// TIA Portal V20 export
DATA_BLOCK "InstShiftmodel"   // DB101
TITLE = Instanz Shiftmodel / InstanceShiftmodel
{ DB_Accessible_From_OPC_UA := 'FALSE' }
AUTHOR : SICAR
FAMILY : Shiftmodel
// Instanz DB / Instance DB
// stored: DBAccessibleFromOPCUA false, InstanceOfName LSicar_Shiftmodel, InstanceOfType FB
"LSicar_Shiftmodel"
   // VAR_OUTPUT
   //    currentShiftCircuitTimes { ExternalAccessible := 'False'; ExternalVisible := 'False'; ExternalWritable := 'False'} : "LSicar_typeShiftmodTime1Shift";
   //    currentShiftTimes { ExternalAccessible := 'False'; ExternalVisible := 'False'; ExternalWritable := 'False'} : "LSicar_typeShiftTimes1Shift";
   // END_VAR
   // VAR_IN_OUT
   //    dateAndTime : "LSicar_typeGlobalDateTime";
   //    shiftTimesHmi : "LSicar_typeShiftmodelHmi";
   //    shiftTimesList : Array[0..10] of "LSicar_typeShiftmodTime1DaySel";
   // END_VAR
   // VAR
   //    statListIdx { ExternalAccessible := 'False'; ExternalVisible := 'False'; ExternalWritable := 'False'} : DInt := 0;
   //    statHmiTimesDay { ExternalAccessible := 'False'; ExternalVisible := 'False'; ExternalWritable := 'False'} : Array[0..7] of "LSicar_typeShiftmodTime1Day";
   //    statHmiSignalsDay { ExternalAccessible := 'False'; ExternalVisible := 'False'; ExternalWritable := 'False'} : Array[0..7] of "LSicar_typeShiftmodSign1Day";
   //    statHmiActualDay { ExternalAccessible := 'False'; ExternalVisible := 'False'; ExternalWritable := 'False'} : USInt := 0;
   //    statShiftTimesListOn { ExternalAccessible := 'False'; ExternalVisible := 'False'; ExternalWritable := 'False'} : Bool := FALSE;
   //    statSummaryHmi { ExternalAccessible := 'False'; ExternalVisible := 'False'; ExternalWritable := 'False'} : "LSicar_typeShiftmodSumHmi";
   //    statHmiShiftmoListindex { ExternalAccessible := 'False'; ExternalVisible := 'False'; ExternalWritable := 'False'} : USInt := 1;
   //    statZeroDay { ExternalAccessible := 'False'; ExternalVisible := 'False'; ExternalWritable := 'False'} : "LSicar_typeShiftmodTime1Day";
   //    statListIndexOld { ExternalAccessible := 'False'; ExternalVisible := 'False'; ExternalWritable := 'False'} : DInt := 1;
   //    statNumberOfWorkDays { ExternalAccessible := 'False'; ExternalVisible := 'False'; ExternalWritable := 'False'} : USInt := 0;
   //    statTimeOfDayActual { ExternalAccessible := 'False'; ExternalVisible := 'False'; ExternalWritable := 'False'} : Time_Of_Day := TOD#00:00:00;
   //    statShiftActual { ExternalAccessible := 'False'; ExternalVisible := 'False'; ExternalWritable := 'False'} : USInt := 0;
   //    statDayCount { ExternalAccessible := 'False'; ExternalVisible := 'False'; ExternalWritable := 'False'} : USInt := 1;
   //    statBreakCount { ExternalAccessible := 'False'; ExternalVisible := 'False'; ExternalWritable := 'False'} : USInt := 0;
   //    statDayChangeNightShift { ExternalAccessible := 'False'; ExternalVisible := 'False'; ExternalWritable := 'False'} : Bool := FALSE;
   //    statDayChangeCircuitTime { ExternalAccessible := 'False'; ExternalVisible := 'False'; ExternalWritable := 'False'} : Bool := FALSE;
   //    statCheckCircuitTime { ExternalAccessible := 'False'; ExternalVisible := 'False'; ExternalWritable := 'False'} : "LSicar_typeShiftCircuitTimes";
   //    statRisEdge { ExternalAccessible := 'False'; ExternalVisible := 'False'; ExternalWritable := 'False'} : "LSicar_typeShiftmodSumHmi";
   //    statPosPulse { ExternalAccessible := 'False'; ExternalVisible := 'False'; ExternalWritable := 'False'} : "LSicar_typeShiftmodSumHmi";
   //    statFalEdge { ExternalAccessible := 'False'; ExternalVisible := 'False'; ExternalWritable := 'False'} : "LSicar_typeShiftmodSumHmi";
   //    statNegPulse { ExternalAccessible := 'False'; ExternalVisible := 'False'; ExternalWritable := 'False'} : "LSicar_typeShiftmodSumHmi";
   //    statTimesAndCircuit { ExternalAccessible := 'False'; ExternalVisible := 'False'; ExternalWritable := 'False'} : "LSicar_typeShiftmodTime1Shift";
   //    statOnlyTimes { ExternalAccessible := 'False'; ExternalVisible := 'False'; ExternalWritable := 'False'} : "LSicar_typeShiftTimes1Shift";
   //    statRisEdgeListOn { ExternalAccessible := 'False'; ExternalVisible := 'False'; ExternalWritable := 'False'} : Bool := FALSE;
   //    statPosPulseListOn { ExternalAccessible := 'False'; ExternalVisible := 'False'; ExternalWritable := 'False'} : Bool := FALSE;
   //    statFalEdgeListOn { ExternalAccessible := 'False'; ExternalVisible := 'False'; ExternalWritable := 'False'} : Bool := FALSE;
   //    statNegPulseListOn { ExternalAccessible := 'False'; ExternalVisible := 'False'; ExternalWritable := 'False'} : Bool := FALSE;
   //    statRisEdgeListChange { ExternalAccessible := 'False'; ExternalVisible := 'False'; ExternalWritable := 'False'} : Bool := FALSE;
   //    statPosPulseListChange { ExternalAccessible := 'False'; ExternalVisible := 'False'; ExternalWritable := 'False'} : Bool := FALSE;
   //    statFirstCycle { ExternalAccessible := 'False'; ExternalVisible := 'False'; ExternalWritable := 'False'} : Bool := TRUE;
   // END_VAR
BEGIN
   currentShiftCircuitTimes.endCircuitTime := TOD#00:00:00;
   currentShiftCircuitTimes.start := TOD#00:00:00;
   currentShiftCircuitTimes.break[0..4].start := TOD#00:00:00;
   currentShiftCircuitTimes.break[0..4].startCircuitTime := TOD#00:00:00;
   currentShiftCircuitTimes.break[0..4].endCircuitTime := TOD#00:00:00;
   currentShiftCircuitTimes.break[0..4].end := TOD#00:00:00;
   currentShiftCircuitTimes.end := TOD#00:00:00;
   currentShiftCircuitTimes.startCircuitTime := TOD#00:00:00;
   currentShiftTimes.start := TOD#00:00:00;
   currentShiftTimes.break[0..4].start := TOD#00:00:00;
   currentShiftTimes.break[0..4].startCircuitTime := TOD#00:00:00;
   currentShiftTimes.break[0..4].endCircuitTime := TOD#00:00:00;
   currentShiftTimes.break[0..4].end := TOD#00:00:00;
   currentShiftTimes.end := TOD#00:00:00;
   statHmiTimesDay[0].shift[0..3].endCircuitTime := TOD#00:00:00;
   statHmiTimesDay[1].shift[0..3].endCircuitTime := TOD#00:00:00;
   statHmiTimesDay[2].shift[0..3].endCircuitTime := TOD#00:00:00;
   statHmiTimesDay[3].shift[0..3].endCircuitTime := TOD#00:00:00;
   statHmiTimesDay[4].shift[0..3].endCircuitTime := TOD#00:00:00;
   statHmiTimesDay[5].shift[0..3].endCircuitTime := TOD#00:00:00;
   statHmiTimesDay[6].shift[0..3].endCircuitTime := TOD#00:00:00;
   statHmiTimesDay[7].shift[0..3].endCircuitTime := TOD#00:00:00;
   statHmiTimesDay[0].shift[0..3].start := TOD#00:00:00;
   statHmiTimesDay[1].shift[0..3].start := TOD#00:00:00;
   statHmiTimesDay[2].shift[0..3].start := TOD#00:00:00;
   statHmiTimesDay[3].shift[0..3].start := TOD#00:00:00;
   statHmiTimesDay[4].shift[0..3].start := TOD#00:00:00;
   statHmiTimesDay[5].shift[0..3].start := TOD#00:00:00;
   statHmiTimesDay[6].shift[0..3].start := TOD#00:00:00;
   statHmiTimesDay[7].shift[0..3].start := TOD#00:00:00;
   statHmiTimesDay[0].shift[0].break[0..4].start := TOD#00:00:00;
   statHmiTimesDay[0].shift[1].break[0..4].start := TOD#00:00:00;
   statHmiTimesDay[0].shift[2].break[0..4].start := TOD#00:00:00;
   statHmiTimesDay[0].shift[3].break[0..4].start := TOD#00:00:00;
   statHmiTimesDay[1].shift[0].break[0..4].start := TOD#00:00:00;
   statHmiTimesDay[1].shift[1].break[0..4].start := TOD#00:00:00;
   statHmiTimesDay[1].shift[2].break[0..4].start := TOD#00:00:00;
   statHmiTimesDay[1].shift[3].break[0..4].start := TOD#00:00:00;
   statHmiTimesDay[2].shift[0].break[0..4].start := TOD#00:00:00;
   statHmiTimesDay[2].shift[1].break[0..4].start := TOD#00:00:00;
   statHmiTimesDay[2].shift[2].break[0..4].start := TOD#00:00:00;
   statHmiTimesDay[2].shift[3].break[0..4].start := TOD#00:00:00;
   statHmiTimesDay[3].shift[0].break[0..4].start := TOD#00:00:00;
   statHmiTimesDay[3].shift[1].break[0..4].start := TOD#00:00:00;
   statHmiTimesDay[3].shift[2].break[0..4].start := TOD#00:00:00;
   statHmiTimesDay[3].shift[3].break[0..4].start := TOD#00:00:00;
   statHmiTimesDay[4].shift[0].break[0..4].start := TOD#00:00:00;
   statHmiTimesDay[4].shift[1].break[0..4].start := TOD#00:00:00;
   statHmiTimesDay[4].shift[2].break[0..4].start := TOD#00:00:00;
   statHmiTimesDay[4].shift[3].break[0..4].start := TOD#00:00:00;
   statHmiTimesDay[5].shift[0].break[0..4].start := TOD#00:00:00;
   statHmiTimesDay[5].shift[1].break[0..4].start := TOD#00:00:00;
   statHmiTimesDay[5].shift[2].break[0..4].start := TOD#00:00:00;
   statHmiTimesDay[5].shift[3].break[0..4].start := TOD#00:00:00;
   statHmiTimesDay[6].shift[0].break[0..4].start := TOD#00:00:00;
   statHmiTimesDay[6].shift[1].break[0..4].start := TOD#00:00:00;
   statHmiTimesDay[6].shift[2].break[0..4].start := TOD#00:00:00;
   statHmiTimesDay[6].shift[3].break[0..4].start := TOD#00:00:00;
   statHmiTimesDay[7].shift[0].break[0..4].start := TOD#00:00:00;
   statHmiTimesDay[7].shift[1].break[0..4].start := TOD#00:00:00;
   statHmiTimesDay[7].shift[2].break[0..4].start := TOD#00:00:00;
   statHmiTimesDay[7].shift[3].break[0..4].start := TOD#00:00:00;
   statHmiTimesDay[0].shift[0].break[0..4].startCircuitTime := TOD#00:00:00;
   statHmiTimesDay[0].shift[1].break[0..4].startCircuitTime := TOD#00:00:00;
   statHmiTimesDay[0].shift[2].break[0..4].startCircuitTime := TOD#00:00:00;
   statHmiTimesDay[0].shift[3].break[0..4].startCircuitTime := TOD#00:00:00;
   statHmiTimesDay[1].shift[0].break[0..4].startCircuitTime := TOD#00:00:00;
   statHmiTimesDay[1].shift[1].break[0..4].startCircuitTime := TOD#00:00:00;
   statHmiTimesDay[1].shift[2].break[0..4].startCircuitTime := TOD#00:00:00;
   statHmiTimesDay[1].shift[3].break[0..4].startCircuitTime := TOD#00:00:00;
   statHmiTimesDay[2].shift[0].break[0..4].startCircuitTime := TOD#00:00:00;
   statHmiTimesDay[2].shift[1].break[0..4].startCircuitTime := TOD#00:00:00;
   statHmiTimesDay[2].shift[2].break[0..4].startCircuitTime := TOD#00:00:00;
   statHmiTimesDay[2].shift[3].break[0..4].startCircuitTime := TOD#00:00:00;
   statHmiTimesDay[3].shift[0].break[0..4].startCircuitTime := TOD#00:00:00;
   statHmiTimesDay[3].shift[1].break[0..4].startCircuitTime := TOD#00:00:00;
   statHmiTimesDay[3].shift[2].break[0..4].startCircuitTime := TOD#00:00:00;
   statHmiTimesDay[3].shift[3].break[0..4].startCircuitTime := TOD#00:00:00;
   statHmiTimesDay[4].shift[0].break[0..4].startCircuitTime := TOD#00:00:00;
   statHmiTimesDay[4].shift[1].break[0..4].startCircuitTime := TOD#00:00:00;
   statHmiTimesDay[4].shift[2].break[0..4].startCircuitTime := TOD#00:00:00;
   statHmiTimesDay[4].shift[3].break[0..4].startCircuitTime := TOD#00:00:00;
   statHmiTimesDay[5].shift[0].break[0..4].startCircuitTime := TOD#00:00:00;
   statHmiTimesDay[5].shift[1].break[0..4].startCircuitTime := TOD#00:00:00;
   statHmiTimesDay[5].shift[2].break[0..4].startCircuitTime := TOD#00:00:00;
   statHmiTimesDay[5].shift[3].break[0..4].startCircuitTime := TOD#00:00:00;
   statHmiTimesDay[6].shift[0].break[0..4].startCircuitTime := TOD#00:00:00;
   statHmiTimesDay[6].shift[1].break[0..4].startCircuitTime := TOD#00:00:00;
   statHmiTimesDay[6].shift[2].break[0..4].startCircuitTime := TOD#00:00:00;
   statHmiTimesDay[6].shift[3].break[0..4].startCircuitTime := TOD#00:00:00;
   statHmiTimesDay[7].shift[0].break[0..4].startCircuitTime := TOD#00:00:00;
   statHmiTimesDay[7].shift[1].break[0..4].startCircuitTime := TOD#00:00:00;
   statHmiTimesDay[7].shift[2].break[0..4].startCircuitTime := TOD#00:00:00;
   statHmiTimesDay[7].shift[3].break[0..4].startCircuitTime := TOD#00:00:00;
   statHmiTimesDay[0].shift[0].break[0..4].endCircuitTime := TOD#00:00:00;
   statHmiTimesDay[0].shift[1].break[0..4].endCircuitTime := TOD#00:00:00;
   statHmiTimesDay[0].shift[2].break[0..4].endCircuitTime := TOD#00:00:00;
   statHmiTimesDay[0].shift[3].break[0..4].endCircuitTime := TOD#00:00:00;
   statHmiTimesDay[1].shift[0].break[0..4].endCircuitTime := TOD#00:00:00;
   statHmiTimesDay[1].shift[1].break[0..4].endCircuitTime := TOD#00:00:00;
   statHmiTimesDay[1].shift[2].break[0..4].endCircuitTime := TOD#00:00:00;
   statHmiTimesDay[1].shift[3].break[0..4].endCircuitTime := TOD#00:00:00;
   statHmiTimesDay[2].shift[0].break[0..4].endCircuitTime := TOD#00:00:00;
   statHmiTimesDay[2].shift[1].break[0..4].endCircuitTime := TOD#00:00:00;
   statHmiTimesDay[2].shift[2].break[0..4].endCircuitTime := TOD#00:00:00;
   statHmiTimesDay[2].shift[3].break[0..4].endCircuitTime := TOD#00:00:00;
   statHmiTimesDay[3].shift[0].break[0..4].endCircuitTime := TOD#00:00:00;
   statHmiTimesDay[3].shift[1].break[0..4].endCircuitTime := TOD#00:00:00;
   statHmiTimesDay[3].shift[2].break[0..4].endCircuitTime := TOD#00:00:00;
   statHmiTimesDay[3].shift[3].break[0..4].endCircuitTime := TOD#00:00:00;
   statHmiTimesDay[4].shift[0].break[0..4].endCircuitTime := TOD#00:00:00;
   statHmiTimesDay[4].shift[1].break[0..4].endCircuitTime := TOD#00:00:00;
   statHmiTimesDay[4].shift[2].break[0..4].endCircuitTime := TOD#00:00:00;
   statHmiTimesDay[4].shift[3].break[0..4].endCircuitTime := TOD#00:00:00;
   statHmiTimesDay[5].shift[0].break[0..4].endCircuitTime := TOD#00:00:00;
   statHmiTimesDay[5].shift[1].break[0..4].endCircuitTime := TOD#00:00:00;
   statHmiTimesDay[5].shift[2].break[0..4].endCircuitTime := TOD#00:00:00;
   statHmiTimesDay[5].shift[3].break[0..4].endCircuitTime := TOD#00:00:00;
   statHmiTimesDay[6].shift[0].break[0..4].endCircuitTime := TOD#00:00:00;
   statHmiTimesDay[6].shift[1].break[0..4].endCircuitTime := TOD#00:00:00;
   statHmiTimesDay[6].shift[2].break[0..4].endCircuitTime := TOD#00:00:00;
   statHmiTimesDay[6].shift[3].break[0..4].endCircuitTime := TOD#00:00:00;
   statHmiTimesDay[7].shift[0].break[0..4].endCircuitTime := TOD#00:00:00;
   statHmiTimesDay[7].shift[1].break[0..4].endCircuitTime := TOD#00:00:00;
   statHmiTimesDay[7].shift[2].break[0..4].endCircuitTime := TOD#00:00:00;
   statHmiTimesDay[7].shift[3].break[0..4].endCircuitTime := TOD#00:00:00;
   statHmiTimesDay[0].shift[0].break[0..4].end := TOD#00:00:00;
   statHmiTimesDay[0].shift[1].break[0..4].end := TOD#00:00:00;
   statHmiTimesDay[0].shift[2].break[0..4].end := TOD#00:00:00;
   statHmiTimesDay[0].shift[3].break[0..4].end := TOD#00:00:00;
   statHmiTimesDay[1].shift[0].break[0..4].end := TOD#00:00:00;
   statHmiTimesDay[1].shift[1].break[0..4].end := TOD#00:00:00;
   statHmiTimesDay[1].shift[2].break[0..4].end := TOD#00:00:00;
   statHmiTimesDay[1].shift[3].break[0..4].end := TOD#00:00:00;
   statHmiTimesDay[2].shift[0].break[0..4].end := TOD#00:00:00;
   statHmiTimesDay[2].shift[1].break[0..4].end := TOD#00:00:00;
   statHmiTimesDay[2].shift[2].break[0..4].end := TOD#00:00:00;
   statHmiTimesDay[2].shift[3].break[0..4].end := TOD#00:00:00;
   statHmiTimesDay[3].shift[0].break[0..4].end := TOD#00:00:00;
   statHmiTimesDay[3].shift[1].break[0..4].end := TOD#00:00:00;
   statHmiTimesDay[3].shift[2].break[0..4].end := TOD#00:00:00;
   statHmiTimesDay[3].shift[3].break[0..4].end := TOD#00:00:00;
   statHmiTimesDay[4].shift[0].break[0..4].end := TOD#00:00:00;
   statHmiTimesDay[4].shift[1].break[0..4].end := TOD#00:00:00;
   statHmiTimesDay[4].shift[2].break[0..4].end := TOD#00:00:00;
   statHmiTimesDay[4].shift[3].break[0..4].end := TOD#00:00:00;
   statHmiTimesDay[5].shift[0].break[0..4].end := TOD#00:00:00;
   statHmiTimesDay[5].shift[1].break[0..4].end := TOD#00:00:00;
   statHmiTimesDay[5].shift[2].break[0..4].end := TOD#00:00:00;
   statHmiTimesDay[5].shift[3].break[0..4].end := TOD#00:00:00;
   statHmiTimesDay[6].shift[0].break[0..4].end := TOD#00:00:00;
   statHmiTimesDay[6].shift[1].break[0..4].end := TOD#00:00:00;
   statHmiTimesDay[6].shift[2].break[0..4].end := TOD#00:00:00;
   statHmiTimesDay[6].shift[3].break[0..4].end := TOD#00:00:00;
   statHmiTimesDay[7].shift[0].break[0..4].end := TOD#00:00:00;
   statHmiTimesDay[7].shift[1].break[0..4].end := TOD#00:00:00;
   statHmiTimesDay[7].shift[2].break[0..4].end := TOD#00:00:00;
   statHmiTimesDay[7].shift[3].break[0..4].end := TOD#00:00:00;
   statHmiTimesDay[0].shift[0..3].end := TOD#00:00:00;
   statHmiTimesDay[1].shift[0..3].end := TOD#00:00:00;
   statHmiTimesDay[2].shift[0..3].end := TOD#00:00:00;
   statHmiTimesDay[3].shift[0..3].end := TOD#00:00:00;
   statHmiTimesDay[4].shift[0..3].end := TOD#00:00:00;
   statHmiTimesDay[5].shift[0..3].end := TOD#00:00:00;
   statHmiTimesDay[6].shift[0..3].end := TOD#00:00:00;
   statHmiTimesDay[7].shift[0..3].end := TOD#00:00:00;
   statHmiTimesDay[0].shift[0..3].startCircuitTime := TOD#00:00:00;
   statHmiTimesDay[1].shift[0..3].startCircuitTime := TOD#00:00:00;
   statHmiTimesDay[2].shift[0..3].startCircuitTime := TOD#00:00:00;
   statHmiTimesDay[3].shift[0..3].startCircuitTime := TOD#00:00:00;
   statHmiTimesDay[4].shift[0..3].startCircuitTime := TOD#00:00:00;
   statHmiTimesDay[5].shift[0..3].startCircuitTime := TOD#00:00:00;
   statHmiTimesDay[6].shift[0..3].startCircuitTime := TOD#00:00:00;
   statHmiTimesDay[7].shift[0..3].startCircuitTime := TOD#00:00:00;
   statHmiSignalsDay[0].shift[0..3].shiftConfig := FALSE;
   statHmiSignalsDay[1].shift[0..3].shiftConfig := FALSE;
   statHmiSignalsDay[2].shift[0..3].shiftConfig := FALSE;
   statHmiSignalsDay[3].shift[0..3].shiftConfig := FALSE;
   statHmiSignalsDay[4].shift[0..3].shiftConfig := FALSE;
   statHmiSignalsDay[5].shift[0..3].shiftConfig := FALSE;
   statHmiSignalsDay[6].shift[0..3].shiftConfig := FALSE;
   statHmiSignalsDay[7].shift[0..3].shiftConfig := FALSE;
   statHmiSignalsDay[0].shift[0..3].shiftActive := FALSE;
   statHmiSignalsDay[1].shift[0..3].shiftActive := FALSE;
   statHmiSignalsDay[2].shift[0..3].shiftActive := FALSE;
   statHmiSignalsDay[3].shift[0..3].shiftActive := FALSE;
   statHmiSignalsDay[4].shift[0..3].shiftActive := FALSE;
   statHmiSignalsDay[5].shift[0..3].shiftActive := FALSE;
   statHmiSignalsDay[6].shift[0..3].shiftActive := FALSE;
   statHmiSignalsDay[7].shift[0..3].shiftActive := FALSE;
   statHmiSignalsDay[0].shift[0..3].shiftEndCirTimeConfig := FALSE;
   statHmiSignalsDay[1].shift[0..3].shiftEndCirTimeConfig := FALSE;
   statHmiSignalsDay[2].shift[0..3].shiftEndCirTimeConfig := FALSE;
   statHmiSignalsDay[3].shift[0..3].shiftEndCirTimeConfig := FALSE;
   statHmiSignalsDay[4].shift[0..3].shiftEndCirTimeConfig := FALSE;
   statHmiSignalsDay[5].shift[0..3].shiftEndCirTimeConfig := FALSE;
   statHmiSignalsDay[6].shift[0..3].shiftEndCirTimeConfig := FALSE;
   statHmiSignalsDay[7].shift[0..3].shiftEndCirTimeConfig := FALSE;
   statHmiSignalsDay[0].shift[0..3].shiftStartCirTimeConfig := FALSE;
   statHmiSignalsDay[1].shift[0..3].shiftStartCirTimeConfig := FALSE;
   statHmiSignalsDay[2].shift[0..3].shiftStartCirTimeConfig := FALSE;
   statHmiSignalsDay[3].shift[0..3].shiftStartCirTimeConfig := FALSE;
   statHmiSignalsDay[4].shift[0..3].shiftStartCirTimeConfig := FALSE;
   statHmiSignalsDay[5].shift[0..3].shiftStartCirTimeConfig := FALSE;
   statHmiSignalsDay[6].shift[0..3].shiftStartCirTimeConfig := FALSE;
   statHmiSignalsDay[7].shift[0..3].shiftStartCirTimeConfig := FALSE;
   statHmiSignalsDay[0].shift[0..3].shiftEndCirTimeActive := FALSE;
   statHmiSignalsDay[1].shift[0..3].shiftEndCirTimeActive := FALSE;
   statHmiSignalsDay[2].shift[0..3].shiftEndCirTimeActive := FALSE;
   statHmiSignalsDay[3].shift[0..3].shiftEndCirTimeActive := FALSE;
   statHmiSignalsDay[4].shift[0..3].shiftEndCirTimeActive := FALSE;
   statHmiSignalsDay[5].shift[0..3].shiftEndCirTimeActive := FALSE;
   statHmiSignalsDay[6].shift[0..3].shiftEndCirTimeActive := FALSE;
   statHmiSignalsDay[7].shift[0..3].shiftEndCirTimeActive := FALSE;
   statHmiSignalsDay[0].shift[0..3].shiftStartCirTimeActive := FALSE;
   statHmiSignalsDay[1].shift[0..3].shiftStartCirTimeActive := FALSE;
   statHmiSignalsDay[2].shift[0..3].shiftStartCirTimeActive := FALSE;
   statHmiSignalsDay[3].shift[0..3].shiftStartCirTimeActive := FALSE;
   statHmiSignalsDay[4].shift[0..3].shiftStartCirTimeActive := FALSE;
   statHmiSignalsDay[5].shift[0..3].shiftStartCirTimeActive := FALSE;
   statHmiSignalsDay[6].shift[0..3].shiftStartCirTimeActive := FALSE;
   statHmiSignalsDay[7].shift[0..3].shiftStartCirTimeActive := FALSE;
   statHmiSignalsDay[0].shift[0..3].shiftSignalsHmi := 16#00;
   statHmiSignalsDay[1].shift[0..3].shiftSignalsHmi := 16#00;
   statHmiSignalsDay[2].shift[0..3].shiftSignalsHmi := 16#00;
   statHmiSignalsDay[3].shift[0..3].shiftSignalsHmi := 16#00;
   statHmiSignalsDay[4].shift[0..3].shiftSignalsHmi := 16#00;
   statHmiSignalsDay[5].shift[0..3].shiftSignalsHmi := 16#00;
   statHmiSignalsDay[6].shift[0..3].shiftSignalsHmi := 16#00;
   statHmiSignalsDay[7].shift[0..3].shiftSignalsHmi := 16#00;
   statHmiSignalsDay[0].shift[0].break[0..4].config := FALSE;
   statHmiSignalsDay[0].shift[1].break[0..4].config := FALSE;
   statHmiSignalsDay[0].shift[2].break[0..4].config := FALSE;
   statHmiSignalsDay[0].shift[3].break[0..4].config := FALSE;
   statHmiSignalsDay[1].shift[0].break[0..4].config := FALSE;
   statHmiSignalsDay[1].shift[1].break[0..4].config := FALSE;
   statHmiSignalsDay[1].shift[2].break[0..4].config := FALSE;
   statHmiSignalsDay[1].shift[3].break[0..4].config := FALSE;
   statHmiSignalsDay[2].shift[0].break[0..4].config := FALSE;
   statHmiSignalsDay[2].shift[1].break[0..4].config := FALSE;
   statHmiSignalsDay[2].shift[2].break[0..4].config := FALSE;
   statHmiSignalsDay[2].shift[3].break[0..4].config := FALSE;
   statHmiSignalsDay[3].shift[0].break[0..4].config := FALSE;
   statHmiSignalsDay[3].shift[1].break[0..4].config := FALSE;
   statHmiSignalsDay[3].shift[2].break[0..4].config := FALSE;
   statHmiSignalsDay[3].shift[3].break[0..4].config := FALSE;
   statHmiSignalsDay[4].shift[0].break[0..4].config := FALSE;
   statHmiSignalsDay[4].shift[1].break[0..4].config := FALSE;
   statHmiSignalsDay[4].shift[2].break[0..4].config := FALSE;
   statHmiSignalsDay[4].shift[3].break[0..4].config := FALSE;
   statHmiSignalsDay[5].shift[0].break[0..4].config := FALSE;
   statHmiSignalsDay[5].shift[1].break[0..4].config := FALSE;
   statHmiSignalsDay[5].shift[2].break[0..4].config := FALSE;
   statHmiSignalsDay[5].shift[3].break[0..4].config := FALSE;
   statHmiSignalsDay[6].shift[0].break[0..4].config := FALSE;
   statHmiSignalsDay[6].shift[1].break[0..4].config := FALSE;
   statHmiSignalsDay[6].shift[2].break[0..4].config := FALSE;
   statHmiSignalsDay[6].shift[3].break[0..4].config := FALSE;
   statHmiSignalsDay[7].shift[0].break[0..4].config := FALSE;
   statHmiSignalsDay[7].shift[1].break[0..4].config := FALSE;
   statHmiSignalsDay[7].shift[2].break[0..4].config := FALSE;
   statHmiSignalsDay[7].shift[3].break[0..4].config := FALSE;
   statHmiSignalsDay[0].shift[0].break[0..4].active := FALSE;
   statHmiSignalsDay[0].shift[1].break[0..4].active := FALSE;
   statHmiSignalsDay[0].shift[2].break[0..4].active := FALSE;
   statHmiSignalsDay[0].shift[3].break[0..4].active := FALSE;
   statHmiSignalsDay[1].shift[0].break[0..4].active := FALSE;
   statHmiSignalsDay[1].shift[1].break[0..4].active := FALSE;
   statHmiSignalsDay[1].shift[2].break[0..4].active := FALSE;
   statHmiSignalsDay[1].shift[3].break[0..4].active := FALSE;
   statHmiSignalsDay[2].shift[0].break[0..4].active := FALSE;
   statHmiSignalsDay[2].shift[1].break[0..4].active := FALSE;
   statHmiSignalsDay[2].shift[2].break[0..4].active := FALSE;
   statHmiSignalsDay[2].shift[3].break[0..4].active := FALSE;
   statHmiSignalsDay[3].shift[0].break[0..4].active := FALSE;
   statHmiSignalsDay[3].shift[1].break[0..4].active := FALSE;
   statHmiSignalsDay[3].shift[2].break[0..4].active := FALSE;
   statHmiSignalsDay[3].shift[3].break[0..4].active := FALSE;
   statHmiSignalsDay[4].shift[0].break[0..4].active := FALSE;
   statHmiSignalsDay[4].shift[1].break[0..4].active := FALSE;
   statHmiSignalsDay[4].shift[2].break[0..4].active := FALSE;
   statHmiSignalsDay[4].shift[3].break[0..4].active := FALSE;
   statHmiSignalsDay[5].shift[0].break[0..4].active := FALSE;
   statHmiSignalsDay[5].shift[1].break[0..4].active := FALSE;
   statHmiSignalsDay[5].shift[2].break[0..4].active := FALSE;
   statHmiSignalsDay[5].shift[3].break[0..4].active := FALSE;
   statHmiSignalsDay[6].shift[0].break[0..4].active := FALSE;
   statHmiSignalsDay[6].shift[1].break[0..4].active := FALSE;
   statHmiSignalsDay[6].shift[2].break[0..4].active := FALSE;
   statHmiSignalsDay[6].shift[3].break[0..4].active := FALSE;
   statHmiSignalsDay[7].shift[0].break[0..4].active := FALSE;
   statHmiSignalsDay[7].shift[1].break[0..4].active := FALSE;
   statHmiSignalsDay[7].shift[2].break[0..4].active := FALSE;
   statHmiSignalsDay[7].shift[3].break[0..4].active := FALSE;
   statHmiSignalsDay[0].shift[0].break[0..4].circuitTimeConfig := FALSE;
   statHmiSignalsDay[0].shift[1].break[0..4].circuitTimeConfig := FALSE;
   statHmiSignalsDay[0].shift[2].break[0..4].circuitTimeConfig := FALSE;
   statHmiSignalsDay[0].shift[3].break[0..4].circuitTimeConfig := FALSE;
   statHmiSignalsDay[1].shift[0].break[0..4].circuitTimeConfig := FALSE;
   statHmiSignalsDay[1].shift[1].break[0..4].circuitTimeConfig := FALSE;
   statHmiSignalsDay[1].shift[2].break[0..4].circuitTimeConfig := FALSE;
   statHmiSignalsDay[1].shift[3].break[0..4].circuitTimeConfig := FALSE;
   statHmiSignalsDay[2].shift[0].break[0..4].circuitTimeConfig := FALSE;
   statHmiSignalsDay[2].shift[1].break[0..4].circuitTimeConfig := FALSE;
   statHmiSignalsDay[2].shift[2].break[0..4].circuitTimeConfig := FALSE;
   statHmiSignalsDay[2].shift[3].break[0..4].circuitTimeConfig := FALSE;
   statHmiSignalsDay[3].shift[0].break[0..4].circuitTimeConfig := FALSE;
   statHmiSignalsDay[3].shift[1].break[0..4].circuitTimeConfig := FALSE;
   statHmiSignalsDay[3].shift[2].break[0..4].circuitTimeConfig := FALSE;
   statHmiSignalsDay[3].shift[3].break[0..4].circuitTimeConfig := FALSE;
   statHmiSignalsDay[4].shift[0].break[0..4].circuitTimeConfig := FALSE;
   statHmiSignalsDay[4].shift[1].break[0..4].circuitTimeConfig := FALSE;
   statHmiSignalsDay[4].shift[2].break[0..4].circuitTimeConfig := FALSE;
   statHmiSignalsDay[4].shift[3].break[0..4].circuitTimeConfig := FALSE;
   statHmiSignalsDay[5].shift[0].break[0..4].circuitTimeConfig := FALSE;
   statHmiSignalsDay[5].shift[1].break[0..4].circuitTimeConfig := FALSE;
   statHmiSignalsDay[5].shift[2].break[0..4].circuitTimeConfig := FALSE;
   statHmiSignalsDay[5].shift[3].break[0..4].circuitTimeConfig := FALSE;
   statHmiSignalsDay[6].shift[0].break[0..4].circuitTimeConfig := FALSE;
   statHmiSignalsDay[6].shift[1].break[0..4].circuitTimeConfig := FALSE;
   statHmiSignalsDay[6].shift[2].break[0..4].circuitTimeConfig := FALSE;
   statHmiSignalsDay[6].shift[3].break[0..4].circuitTimeConfig := FALSE;
   statHmiSignalsDay[7].shift[0].break[0..4].circuitTimeConfig := FALSE;
   statHmiSignalsDay[7].shift[1].break[0..4].circuitTimeConfig := FALSE;
   statHmiSignalsDay[7].shift[2].break[0..4].circuitTimeConfig := FALSE;
   statHmiSignalsDay[7].shift[3].break[0..4].circuitTimeConfig := FALSE;
   statHmiSignalsDay[0].shift[0].break[0..4].circuitTimeActive := FALSE;
   statHmiSignalsDay[0].shift[1].break[0..4].circuitTimeActive := FALSE;
   statHmiSignalsDay[0].shift[2].break[0..4].circuitTimeActive := FALSE;
   statHmiSignalsDay[0].shift[3].break[0..4].circuitTimeActive := FALSE;
   statHmiSignalsDay[1].shift[0].break[0..4].circuitTimeActive := FALSE;
   statHmiSignalsDay[1].shift[1].break[0..4].circuitTimeActive := FALSE;
   statHmiSignalsDay[1].shift[2].break[0..4].circuitTimeActive := FALSE;
   statHmiSignalsDay[1].shift[3].break[0..4].circuitTimeActive := FALSE;
   statHmiSignalsDay[2].shift[0].break[0..4].circuitTimeActive := FALSE;
   statHmiSignalsDay[2].shift[1].break[0..4].circuitTimeActive := FALSE;
   statHmiSignalsDay[2].shift[2].break[0..4].circuitTimeActive := FALSE;
   statHmiSignalsDay[2].shift[3].break[0..4].circuitTimeActive := FALSE;
   statHmiSignalsDay[3].shift[0].break[0..4].circuitTimeActive := FALSE;
   statHmiSignalsDay[3].shift[1].break[0..4].circuitTimeActive := FALSE;
   statHmiSignalsDay[3].shift[2].break[0..4].circuitTimeActive := FALSE;
   statHmiSignalsDay[3].shift[3].break[0..4].circuitTimeActive := FALSE;
   statHmiSignalsDay[4].shift[0].break[0..4].circuitTimeActive := FALSE;
   statHmiSignalsDay[4].shift[1].break[0..4].circuitTimeActive := FALSE;
   statHmiSignalsDay[4].shift[2].break[0..4].circuitTimeActive := FALSE;
   statHmiSignalsDay[4].shift[3].break[0..4].circuitTimeActive := FALSE;
   statHmiSignalsDay[5].shift[0].break[0..4].circuitTimeActive := FALSE;
   statHmiSignalsDay[5].shift[1].break[0..4].circuitTimeActive := FALSE;
   statHmiSignalsDay[5].shift[2].break[0..4].circuitTimeActive := FALSE;
   statHmiSignalsDay[5].shift[3].break[0..4].circuitTimeActive := FALSE;
   statHmiSignalsDay[6].shift[0].break[0..4].circuitTimeActive := FALSE;
   statHmiSignalsDay[6].shift[1].break[0..4].circuitTimeActive := FALSE;
   statHmiSignalsDay[6].shift[2].break[0..4].circuitTimeActive := FALSE;
   statHmiSignalsDay[6].shift[3].break[0..4].circuitTimeActive := FALSE;
   statHmiSignalsDay[7].shift[0].break[0..4].circuitTimeActive := FALSE;
   statHmiSignalsDay[7].shift[1].break[0..4].circuitTimeActive := FALSE;
   statHmiSignalsDay[7].shift[2].break[0..4].circuitTimeActive := FALSE;
   statHmiSignalsDay[7].shift[3].break[0..4].circuitTimeActive := FALSE;
   statHmiSignalsDay[0].shift[0..3].breakSignalsHmi := 16#0000;
   statHmiSignalsDay[1].shift[0..3].breakSignalsHmi := 16#0000;
   statHmiSignalsDay[2].shift[0..3].breakSignalsHmi := 16#0000;
   statHmiSignalsDay[3].shift[0..3].breakSignalsHmi := 16#0000;
   statHmiSignalsDay[4].shift[0..3].breakSignalsHmi := 16#0000;
   statHmiSignalsDay[5].shift[0..3].breakSignalsHmi := 16#0000;
   statHmiSignalsDay[6].shift[0..3].breakSignalsHmi := 16#0000;
   statHmiSignalsDay[7].shift[0..3].breakSignalsHmi := 16#0000;
   statHmiSignalsDay[0..7].shiftsPerDay := 0;
   statSummaryHmi.earlyShiftActive := FALSE;
   statSummaryHmi.lateShiftActive := FALSE;
   statSummaryHmi.nightShiftActive := FALSE;
   statSummaryHmi.breakInShiftActive := FALSE;
   statSummaryHmi.breakBetweenShiftAct := FALSE;
   statSummaryHmi.breakActive := FALSE;
   statSummaryHmi.circuitTimeInShiftAct := FALSE;
   statSummaryHmi.circuitTimeBetwShiftAct := FALSE;
   statSummaryHmi.circuitTimeActive := FALSE;
   statSummaryHmi.noOfWorkdays := 0;
   statSummaryHmi.workdays[0..7] := FALSE;
   statZeroDay.shift[0..3].endCircuitTime := TOD#00:00:00;
   statZeroDay.shift[0..3].start := TOD#00:00:00;
   statZeroDay.shift[0].break[0..4].start := TOD#00:00:00;
   statZeroDay.shift[1].break[0..4].start := TOD#00:00:00;
   statZeroDay.shift[2].break[0..4].start := TOD#00:00:00;
   statZeroDay.shift[3].break[0..4].start := TOD#00:00:00;
   statZeroDay.shift[0].break[0..4].startCircuitTime := TOD#00:00:00;
   statZeroDay.shift[1].break[0..4].startCircuitTime := TOD#00:00:00;
   statZeroDay.shift[2].break[0..4].startCircuitTime := TOD#00:00:00;
   statZeroDay.shift[3].break[0..4].startCircuitTime := TOD#00:00:00;
   statZeroDay.shift[0].break[0..4].endCircuitTime := TOD#00:00:00;
   statZeroDay.shift[1].break[0..4].endCircuitTime := TOD#00:00:00;
   statZeroDay.shift[2].break[0..4].endCircuitTime := TOD#00:00:00;
   statZeroDay.shift[3].break[0..4].endCircuitTime := TOD#00:00:00;
   statZeroDay.shift[0].break[0..4].end := TOD#00:00:00;
   statZeroDay.shift[1].break[0..4].end := TOD#00:00:00;
   statZeroDay.shift[2].break[0..4].end := TOD#00:00:00;
   statZeroDay.shift[3].break[0..4].end := TOD#00:00:00;
   statZeroDay.shift[0..3].end := TOD#00:00:00;
   statZeroDay.shift[0..3].startCircuitTime := TOD#00:00:00;
   statCheckCircuitTime.startTime := TOD#00:00:00;
   statCheckCircuitTime.fromDay := 1;
   statCheckCircuitTime.fromShift := 1;
   statCheckCircuitTime.endTime := TOD#00:00:00;
   statCheckCircuitTime.toDay := 1;
   statCheckCircuitTime.toShift := 1;
   statRisEdge.earlyShiftActive := FALSE;
   statRisEdge.lateShiftActive := FALSE;
   statRisEdge.nightShiftActive := FALSE;
   statRisEdge.breakInShiftActive := FALSE;
   statRisEdge.breakBetweenShiftAct := FALSE;
   statRisEdge.breakActive := FALSE;
   statRisEdge.circuitTimeInShiftAct := FALSE;
   statRisEdge.circuitTimeBetwShiftAct := FALSE;
   statRisEdge.circuitTimeActive := FALSE;
   statRisEdge.noOfWorkdays := 0;
   statRisEdge.workdays[0..7] := FALSE;
   statPosPulse.earlyShiftActive := FALSE;
   statPosPulse.lateShiftActive := FALSE;
   statPosPulse.nightShiftActive := FALSE;
   statPosPulse.breakInShiftActive := FALSE;
   statPosPulse.breakBetweenShiftAct := FALSE;
   statPosPulse.breakActive := FALSE;
   statPosPulse.circuitTimeInShiftAct := FALSE;
   statPosPulse.circuitTimeBetwShiftAct := FALSE;
   statPosPulse.circuitTimeActive := FALSE;
   statPosPulse.noOfWorkdays := 0;
   statPosPulse.workdays[0..7] := FALSE;
   statFalEdge.earlyShiftActive := FALSE;
   statFalEdge.lateShiftActive := FALSE;
   statFalEdge.nightShiftActive := FALSE;
   statFalEdge.breakInShiftActive := FALSE;
   statFalEdge.breakBetweenShiftAct := FALSE;
   statFalEdge.breakActive := FALSE;
   statFalEdge.circuitTimeInShiftAct := FALSE;
   statFalEdge.circuitTimeBetwShiftAct := FALSE;
   statFalEdge.circuitTimeActive := FALSE;
   statFalEdge.noOfWorkdays := 0;
   statFalEdge.workdays[0..7] := FALSE;
   statNegPulse.earlyShiftActive := FALSE;
   statNegPulse.lateShiftActive := FALSE;
   statNegPulse.nightShiftActive := FALSE;
   statNegPulse.breakInShiftActive := FALSE;
   statNegPulse.breakBetweenShiftAct := FALSE;
   statNegPulse.breakActive := FALSE;
   statNegPulse.circuitTimeInShiftAct := FALSE;
   statNegPulse.circuitTimeBetwShiftAct := FALSE;
   statNegPulse.circuitTimeActive := FALSE;
   statNegPulse.noOfWorkdays := 0;
   statNegPulse.workdays[0..7] := FALSE;
   statTimesAndCircuit.endCircuitTime := TOD#00:00:00;
   statTimesAndCircuit.start := TOD#00:00:00;
   statTimesAndCircuit.break[0..4].start := TOD#00:00:00;
   statTimesAndCircuit.break[0..4].startCircuitTime := TOD#00:00:00;
   statTimesAndCircuit.break[0..4].endCircuitTime := TOD#00:00:00;
   statTimesAndCircuit.break[0..4].end := TOD#00:00:00;
   statTimesAndCircuit.end := TOD#00:00:00;
   statTimesAndCircuit.startCircuitTime := TOD#00:00:00;
   statOnlyTimes.start := TOD#00:00:00;
   statOnlyTimes.break[0..4].start := TOD#00:00:00;
   statOnlyTimes.break[0..4].startCircuitTime := TOD#00:00:00;
   statOnlyTimes.break[0..4].endCircuitTime := TOD#00:00:00;
   statOnlyTimes.break[0..4].end := TOD#00:00:00;
   statOnlyTimes.end := TOD#00:00:00;
END_DATA_BLOCK
